// TIA Portal V19 export
VAR_GLOBAL   // PLC tag table "Program_CONST"
END_VAR
VAR_GLOBAL CONSTANT   // user constants
   PPRG_TOTAL_ARCHIVE_ITEMS : Int := 2000;
   HMI_LIST_ITEMS : Int := 15;
   PPRF_TOTAL_ARCHIVE_ITEMS : Int := 100;
END_VAR
